RoboDK station: BakkeSim.rdk

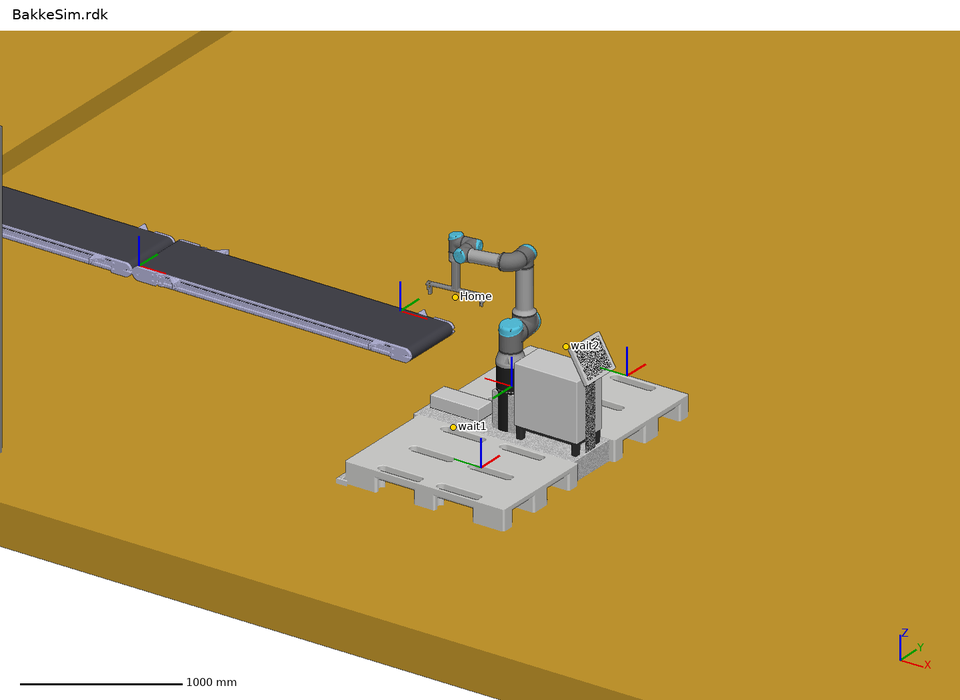
[picture v0: the station drawn from its stored meshes, robots at their saved joint values, targets as dots, program paths as lines]
Station BakkeSim. Poses are relative to the parent item; angles as X-Y-Z fixed-axis rotations.
  - object AVD_Sjokko_SjokkPall2018_Utsnitt at (-66000, -40000, 0) mm, size 13177.1 x 13563.5 x 2830.1 mm, geometry from AVD_Sjokko_SjokkPall2018_Utsnitt.iges
  - frame Conveyor Belt Base at (-8190, -5480, 600) mm
    - robot Conveyor Belt: 1 axes
        modified DH rows (alpha deg, a mm, theta deg, d mm): 0, 0, 0, 0 linear
        base shift (0, 0, 0) mm, rotated rx 0 ry 90 rz 0 deg
        joint limits [-500000] to [500000]; home [0]; saved at [2601.542]
  - frame Conveyor Belt Base at (-6090, -5480, 600) mm
    - robot Conveyor Belt: 1 axes
        modified DH rows (alpha deg, a mm, theta deg, d mm): 0, 0, 0, 0 linear
        base shift (0, 0, 0) mm, rotated rx 0 ry 90 rz 0 deg
        joint limits [-500000] to [500000]; home [0]; saved at [0]
  - object main041119-v2-v2 at (0, 0, 0) mm, size 2050.3 x 1281 x 896.7 mm, geometry from main041119-v2-v2.step
    - object pallPlast-v2 at (-30, 0, 0) mm, size 800 x 1200 x 150 mm, geometry from pallPlast-v2.step
  - object pallPlast-v2 at (-30, -1190, 0) mm, size 800 x 1200 x 150 mm, geometry from pallPlast-v2.step
  - frame UR16e Base at (-3450, -5250, 420) mm, rotated rx 0 ry 0 rz 180 deg
    - target Home (Cartesian target) at (501.54, -113.45, 422.55) mm, rotated rx -180 ry 0 rz -83.47 deg; joints [-148.47, -90, -90, -90, 90, 0] of UR16e
    - frame Pickframe at (830, 10, 290) mm, rotated rx 0 ry 0 rz 180 deg
    - frame placeFrame1 at (-320, 790, -150) mm, rotated rx 0 ry 0 rz -90 deg
    - target wait1 (Cartesian target) at (-30.74, 670.56, -4.96) mm, rotated rx -179.95 ry 0.02 rz -0.09 deg; joints [-46.78, -132.764, -103.803, -33.382, 90, 18.31] of UR16e
    - frame placeFrame2 at (-320, -780, -150) mm, rotated rx 0 ry 0 rz -90 deg
    - target wait2 (Cartesian target) at (52.64, -659.98, -4.81) mm, rotated rx -179.93 ry 0.02 rz -179.06 deg; joints [-225.76, -134.43, -104.03, -31.47, 90, 18.3] of UR16e
  - frame Heis Base at (-3450, -5250, 420) mm, rotated rx 0 ry 0 rz 180 deg
    - robot Heis: 1 axes
        modified DH rows (alpha deg, a mm, theta deg, d mm): 0, 0, 0, 0 linear
        base shift (0, 0, 0) mm, rotated rx 0 ry 0 rz 90 deg
        joint limits [0] to [900]; home [0]; saved at [6.08]
      - object stolpe-v2 at (5, 5, -540) mm, size 180 x 180 x 700 mm, geometry from stolpe-v2.step
      - robot UR16e: 6 axes, payload 16 kg, reach 900 mm, repeatability 0.05 mm, weight 33.1 kg
          modified DH rows (alpha deg, a mm, theta deg, d mm): 0, 0, 0, 180.7; 90, 0, 180, 0; 0, 478.4, 0, 0; 0, 360, 0, 174.15; -90, 0, 0, 119.85; 90, 0, 180, 116.55
          base shift (5, 5, 160) mm, rotated rx 0 ry 0 rz 155 deg
          joint limits [-360, -360, -360, -360, -360, -360] to [360, 360, 360, 360, 360, 360]; home [0, -90, -90, 0, 90, 0]; saved at [-148.47, -90.043, -92.517, -87.44, 90, 0]
        - tool gripperStorbox-v3201119, TCP at (0, 0, 270) mm, size 397.9 x 90 x 286 mm, geometry from gripperStorbox-v3201119.step
    - target Target 1 (Cartesian target) at (0, 0, 6.08) mm; joints [6.08, 0, 0, 0, 0, 0] of Heis
  - object storbox-v2 at (-60, 110, -120) mm, size 385 x 533.3 x 120.2 mm, geometry from storbox-v2.step
